// Mitsubishi GX Works2 project: TIMER   PLC: Q03UDV

PROGRAM MAIN
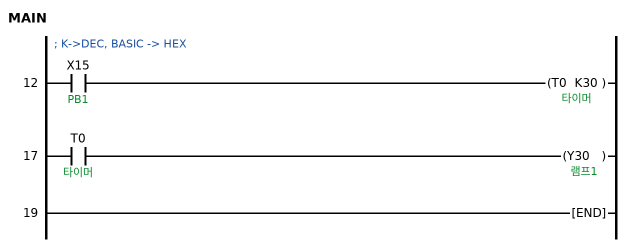
; K->DEC, BASIC -> HEX
12    LD      X15  ; PB1
      OUT     T0 K30  ; 타이머
17    LD      T0  ; 타이머
      OUT     Y30  ; 램프1
19    END
END_PROGRAM
